FUNCTION_BLOCK FB_Interlock
VAR_INPUT
	i_bInterlocked : BOOL;
END_VAR
VAR
	s_bInterlocked : BOOL;
	s_sReason : STRING;
END_VAR


s_bInterlocked := i_bInterlocked;

PROPERTY PUBLIC p_bInterlocked : BOOL
GET

p_bInterlocked := s_bInterlocked;
END_GET
END_PROPERTY

PROPERTY PUBLIC p_sReason : STRING
GET

p_sReason := s_sReason;
END_GET
SET

s_sReason := p_sReason;
END_SET
END_PROPERTY

END_FUNCTION_BLOCK

(* stored: Version 1.1.0.1, ProductVersion 3.1.4024.12
   POU FB_Interlock: Id {4b1f4aa1-d5c6-4fba-8255-b2fd1cb501aa}, SpecialFunc None
   Property p_bInterlocked: Id {4cbb4d8a-b269-4207-b907-0e7be8284474}
   Get Get: Id {5969b6fb-152b-480d-ba12-b6a924ac9874}
   Property p_sReason: Id {b38bc880-c347-4b9a-abef-94cb5823b953}
   Get Get: Id {aac7f1de-102d-4008-bd59-863e8437a056}
   Set Set: Id {d3cd87a1-2189-41fd-98d4-b8a3e8d32560} *)
